TYPE FW212CAttenuationFilterConfig EXTENDS DeviceConfiguration :
STRUCT
	SerialCommunication : SerialCommunication;
END_STRUCT
END_TYPE

(* stored: Version 1.1.0.1, ProductVersion 3.1.4024.4
   DUT FW212CAttenuationFilterConfig: Id {2fe81528-a1c8-4c73-a8e2-03ee61b1bcac} *)
